(* PLC project PLC, Beckhoff Automation GmbH TwinCAT PLC Control 3.5.20.60 *)
(* stored: creationDateTime 2026-07-21T08:44:17.4518911, modificationDateTime 2026-07-21T08:44:17.4548882 *)

TYPE ST_ADS_API_ScadaViewerApp :

STRUCT

	In			:	ST_ADS_API_ScadaViewerApp_PLC_In;		// |1| Vstupní data od PC aplikace
	Out			:	ST_ADS_API_ScadaViewerApp_PLC_Out;		// |2| Výstupní data do PC aplikace
	
END_STRUCT

END_TYPE
